# EPICS alarm handler configuration: caQtDM_UnitTests/tst_qtcontrols/fixtures/alh/include_main.alhConfig
GROUP NULL TOP
CHANNEL TOP top:ch
INCLUDE TOP include_sub.alhConfig
GROUP TOP AFTER
INCLUDE TOP missing_file.alhConfig
INCLUDE NULL include_loop.alhConfig
